// TwinCAT 3 PLC project MultiTankCoolingSystem
// ProgramVersion: 3.1.4024.0
// libraries:
//   Tc2_Standard, * (Beckhoff Automation GmbH)
//   Tc2_System, * (Beckhoff Automation GmbH)
//   Tc3_Module, * (Beckhoff Automation GmbH)
// project tree:
//   DUTs/ ST_Tank.TcDUT
//   GVLs/ GVL.TcGVL
//   / PlcTask.TcTTO
//   POUs/ FB_TankController.TcPOU, F_CheckAlarm.TcPOU, F_CoolTank.TcPOU, I_TankController.TcIO, MAIN.TcPOU, TransferChemical.TcPOU
// real-time tasks:
//   TASK PlcTask: cycle T#10ms, priority 20, ADS port 350
//   TASK PlcTask1: cycle T#10ms, priority 21, ADS port 351
//   TASK PlcTask2: cycle T#10ms, priority 22, ADS port 352

CONFIGURATION MultiTankCoolingSystem
    RESOURCE PLC ON TwinCAT3
        TASK PlcTask(INTERVAL := T#10ms, PRIORITY := 21);
        PROGRAM MAIN WITH PlcTask : MAIN;
    END_RESOURCE
END_CONFIGURATION

// ---- DUTs/ST_Tank.TcDUT
TYPE ST_Tank :
STRUCT
	nId : INT;
	fTemperature : REAL;
	fLevel : REAL;
	bTemperatureAlarm : BOOL;
	bLevelAlarm : BOOL;
END_STRUCT
END_TYPE

// ---- GVLs/GVL.TcGVL
{attribute 'qualified_only'}
VAR_GLOBAL CONSTANT
	fMaxTemperature : REAL := 80;
	fMaxLevelPercentage: REAL := 90.0;
	fCoolingSpeed : REAL := 3;
	fRequiredTemperature: REAL := 50.0;
	fRequiredLevel : REAL := 30;
	fTransferSpeed : REAL := 10;
	fProcessLevel : REAL := 10;
	fProcessTemperature : REAL := 5;
END_VAR

// ---- POUs/I_TankController.TcIO
INTERFACE I_TankController

METHOD ApplyCooling 
VAR_INPUT
END_VAR
END_METHOD

METHOD CheckSafety
VAR_INPUT
END_VAR
END_METHOD

METHOD DispenseChemical 
VAR_INPUT
END_VAR
END_METHOD

END_INTERFACE

// ---- POUs/MAIN.TcPOU
PROGRAM MAIN
VAR
	stTank1 : ST_Tank := (nId := 101,fTemperature := 80.3, fLevel := 80 );
	stTank2 : ST_Tank  := (nId := 102,fTemperature := 72.5, fLevel := 70 );
	stTank3 : ST_Tank  := (nId := 103,fTemperature := 90.8, fLevel := 95 );
	
	fbController : FB_TankController;
	
	bStart : bool;
END_VAR

IF bStart THEN
	fbController(stTank := stTank1);
	fbController(stTank := stTank2);
	fbController(stTank := stTank3);
	bStart := FALSE;
END_IF

END_PROGRAM

// ---- POUs/FB_TankController.TcPOU
FUNCTION_BLOCK FB_TankController IMPLEMENTS I_TankController
VAR_IN_OUT
	stTank : ST_Tank;
END_VAR
VAR
END_VAR


IF __ISVALIDREF(stTank) THEN
	CheckSafety();
	IF (stTank.bTemperatureAlarm) OR (stTank.bLevelAlarm) THEN
		IF stTank.bTemperatureAlarm THEN
			ApplyCooling();
			RETURN;
		END_IF
		IF stTank.bLevelAlarm THEN
			DispenseChemical();
		END_IF
	END_IF
	IF NOT (stTank.bTemperatureAlarm) AND NOT (stTank.bLevelAlarm) THEN
		TankProcessing();
	END_IF
END_IF

{warning 'add method implementation '}
METHOD ApplyCooling : BOOL

F_CoolTank(stTank);
END_METHOD

{warning 'add method implementation '}
METHOD CheckSafety : BOOL
F_CheckAlarm( pTank := ADR(stTank) )
END_METHOD

METHOD DispenseChemical : BOOL
VAR_INPUT
END_VAR
IF stTank.bLevelAlarm THEN
	TransferChemical( pTank := ADR(stTank) );
END_IF
END_METHOD

METHOD TankProcessing : BOOL
VAR_INPUT
END_VAR
stTank.fTemperature := stTank.fTemperature + GVL.fProcessTemperature;
stTank.fLevel := stTank.fLevel + GVL.fProcessLevel;
END_METHOD

END_FUNCTION_BLOCK

// ---- POUs/F_CoolTank.TcPOU
FUNCTION F_CoolTank : BOOL
VAR_INPUT
	rTank : REFERENCE TO ST_Tank;
END_VAR
VAR
	
END_VAR

IF __ISVALIDREF(rTank) THEN
	IF rTank.fTemperature > GVL.fRequiredTemperature THEN
		rTank.fTemperature := rTank.fTemperature - GVL.fCoolingSpeed;
	ELSE
		rTank.bTemperatureAlarm := FALSE;
	END_IF
END_IF

END_FUNCTION

// ---- POUs/F_CheckAlarm.TcPOU
FUNCTION F_CheckAlarm : BOOL
VAR_INPUT
	pTank : POINTER TO ST_Tank;
END_VAR
VAR
	fLevel : REAL := pTank^.fLevel;
	fTemperature : REAL := pTank^.fTemperature;
END_VAR


IF pTank <> 0 THEN
	IF fLevel > GVL.fMaxLevelPercentage THEN
		pTank^.bLevelAlarm := TRUE;
	END_IF
	IF fTemperature > GVL.fMaxTemperature THEN
		pTank^.bTemperatureAlarm := TRUE;
	END_IF
END_IF

END_FUNCTION

// ---- POUs/TransferChemical.TcPOU
FUNCTION TransferChemical : BOOL
VAR_INPUT
	pTank : POINTER TO ST_Tank;
END_VAR
VAR
	
END_VAR

IF pTank <> 0 THEN
	IF pTank^.fLevel > GVL.fRequiredLevel THEN
		pTank^.fLevel := pTank^.fLevel - GVL.fTransferSpeed;
	ELSE
		PTank^.bLevelAlarm := FALSE;
	END_IF
END_IF

END_FUNCTION
